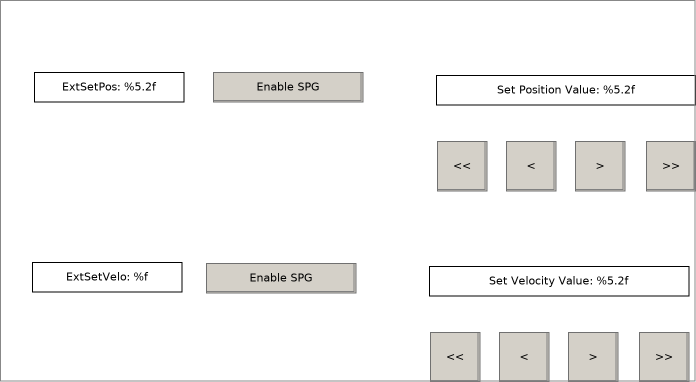
VISUALIZATION Basic_ESPG  // 696x382
    Rectangle (34,72 150x30), "ExtSetPos: %5.2f", text variable: BasicESPG_Position.Basic_Axis.PlcToNc.ExtSetPos
    Rectangle (32,262 150x30), "ExtSetVelo: %f", text variable: BasicESPG_Velocity.Basic_Axis.PlcToNc.ExtSetVelo
    Button (213,72 150x30), "Enable SPG"
        toggle BasicESPG_Position.Execute
    Rectangle (436,75 260x30), "Set Position Value: %5.2f", text variable: BasicESPG_Position.NextIncrementalPosition
    Button (575,141 50x50), ">"
        toggle BasicESPG_Position.Inc1
    Button (646,141 50x50), ">>"
        toggle BasicESPG_Position.Inc10
    Button (506,141 50x50), "<"
        toggle BasicESPG_Position.Dec1
    Button (437,141 50x50), "<<"
        toggle BasicESPG_Position.Dec10
    Button (206,263 150x30), "Enable SPG"
        toggle BasicESPG_Velocity.Execute
    Rectangle (429,266 260x30), "Set Velocity Value: %5.2f", text variable: BasicESPG_Velocity.NextIncrementalVelocity
    Button (568,332 50x50), ">"
        toggle BasicESPG_Velocity.Inc1
    Button (639,332 50x50), ">>"
        toggle BasicESPG_Velocity.Inc10
    Button (499,332 50x50), "<"
        toggle BasicESPG_Velocity.Dec1
    Button (430,332 50x50), "<<"
        toggle BasicESPG_Velocity.Dec10
END_VISUALIZATION

(* stored: Version 1.1.0.1, ProductVersion 3.1.4024.12
   Visu Basic_ESPG: Id {0dd62b7e-23cd-47c4-9610-8651e22cf8e3} *)
